(* Logix 5000 project; controller simObli1_rev_1 Emulate 5570 rev 32.11; software revision 32.02 *)

TASK MainTask (continuous, watchdog 500 ms) : MainProgram, Alarmer, MS1_2_Function
TASK simulering (periodic, rate 10 ms, priority 10, watchdog 500 ms) : mainSim
TASK Temp_regulering (periodic, rate 100 ms, priority 10, watchdog 500 ms) : Heat_reg
TASK Tryk_regulering (periodic, rate 500 ms, priority 10, watchdog 500 ms) : Tryk_regulering_PID

MODULES
   Local : Emulate 5570 (ICP 3, rev 32.11)
END_MODULES

TYPE SP :   // De forskellige setpunkter
STRUCT
   Tryk : REAL;   // Tryk regulering
END_STRUCT
END_TYPE

ADD_ON_INSTRUCTION Add_three_Numbers   (* revision 1.0 *)
VAR_INPUT
   nr1 : REAL; {required}
   nr2 : REAL; {required}
   nr3 : REAL; {required}
END_VAR
VAR_OUTPUT
   nr4 : REAL; {access Read Only, required}
END_VAR
VAR
   ADD_01 : FBD_MATH; {access None}
   ADD_02 : FBD_MATH; {access None}
   __l3847ED3F9690BCDD : REAL; {access None}
   __lAC4B0D8890163B21 : REAL; {access None}
   __l5BA8AF029BD9C521 : REAL; {access None}
END_VAR

ROUTINE Logic   (* function block diagram *)
   SHEET 1
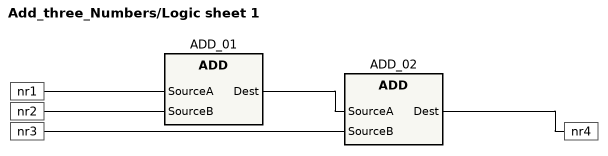
   ADD_01 : ADD(SourceA := nr1, SourceB := nr2);
   ADD_02 : ADD(SourceA := ADD_01.Dest, SourceB := nr3);
   nr4 := ADD_02.Dest;
END_ROUTINE
END_ADD_ON_INSTRUCTION

ADD_ON_INSTRUCTION IMC_Sim   (* revision 1.0 *)
VAR_INPUT
   IMC_CV : REAL; {required}
   IMC_Sim_Reset : BOOL;
   PosNegGain : BOOL;
   DeadTime : REAL := 40.0;
   Lag1 : REAL := 20.0;
   Lag2 : REAL := 20.0;
END_VAR
VAR_OUTPUT
   IMC_PV : REAL; {access Read Only, required}
END_VAR
VAR
   LDLG_01 : LEAD_LAG := (Lag := 30.0, Gain := 1.0, RTSTime := 1);
   LDLG_02 : LEAD_LAG := (Lag := 5.0, Gain := 1.0, RTSTime := 1);
   DEDT_01 : DEADTIME := (Deadtime := 5.0, Gain := 1.0, RTSTime := 1);
   DAIMC : REAL[500];
   SEL_01 : SELECT := (In1 := 1.0, In2 := -1.0);
   SUB_01 : FBD_MATH := (SourceA := 100.0);
   __l19C25824DC418C7C : REAL; {access None}
   __l063CFE09B5704E10 : REAL; {access None}
   __l53C0B5411D4AFA12 : BOOL; {access None}
   __l688BFD8304F18446 : REAL; {access None}
   __l9A341ECD8A034AB4 : REAL; {access None}
   __l887D6C7A4353A221 : BOOL; {access None}
END_VAR

ROUTINE Logic   (* function block diagram *)
   SHEET 1
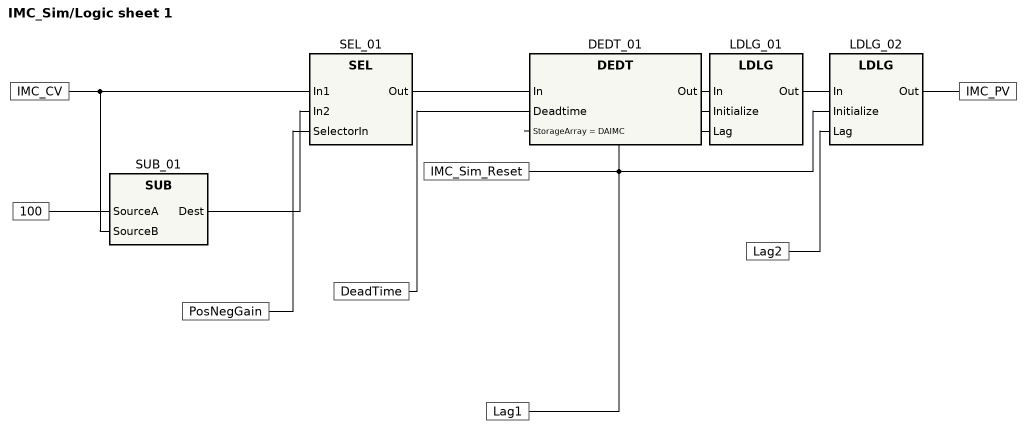
   SUB_01 : SUB(SourceA := 100, SourceB := IMC_CV);
   SEL_01 : SEL(In1 := IMC_CV, In2 := SUB_01.Dest, SelectorIn := PosNegGain);
   DEDT_01 : DEDT(In := SEL_01.Out, Deadtime := DeadTime, StorageArray := DAIMC);
   LDLG_01 : LDLG(In := DEDT_01.Out, Initialize := IMC_Sim_Reset, Lag := Lag1);
   LDLG_02 : LDLG(In := LDLG_01.Out, Initialize := IMC_Sim_Reset, Lag := Lag2);
   IMC_PV := LDLG_02.Out;
END_ROUTINE
END_ADD_ON_INSTRUCTION

ADD_ON_INSTRUCTION Invers_Direkte   (* revision 1.0 *)
VAR_INPUT
   PV : REAL; {required}
   SP : REAL; {required}
END_VAR
VAR_OUTPUT
   fejl_e : REAL; {access None, visible}
END_VAR
VAR_INPUT
   Invers_Direkte : BOOL; {access None, required}
END_VAR
VAR
   SUB_01 : FBD_MATH; {access None}
   SUB_02 : FBD_MATH; {access None}
   SEL_01 : SELECT; {access None}
   Invers : FBD_MATH; {access None}
   Direkte : FBD_MATH; {access None}
   __lF2B22BFB3DCEA4AD : BOOL; {access None}
   __l05D6903D8B432843 : REAL; {access None}
   __lC89B16A93BBA0745 : REAL; {access None}
END_VAR

ROUTINE Logic   (* function block diagram *)
   SHEET 1
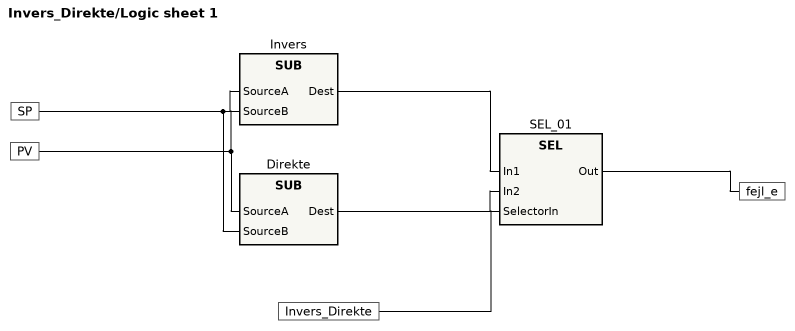
   Invers : SUB(SourceA := SP, SourceB := PV);
   Direkte : SUB(SourceA := PV, SourceB := SP);
   SEL_01 : SEL(In1 := Invers.Dest, In2 := Direkte.Dest, SelectorIn := Invers_Direkte);
   fejl_e := SEL_01.Out;
END_ROUTINE
END_ADD_ON_INSTRUCTION

ADD_ON_INSTRUCTION PID_regulator   (* revision 1.0 *)
VAR_INPUT
   SP : REAL; {access None, visible}
   PV : REAL; {access None, visible}
   Kp : REAL; {access None, visible}
   Ki : REAL; {access None, visible}
   Kd : REAL; {visible}
   U0 : REAL; {visible}
   U_man : REAL; {visible}
END_VAR
VAR_OUTPUT
   CV : REAL; {access Read Only, visible}
END_VAR
VAR_INPUT
   Invers_Direkte : BOOL; {access None, visible}
   Manuel_Auto : BOOL; {access None, visible}
   Reset : BOOL; {visible}
END_VAR
VAR
   Add_three_Numbers_01 : Add_three_Numbers; {access None}
   Invers_Direkte_01 : Invers_Direkte; {access None}
   ADD_02 : FBD_MATH := (SourceA := 23.71752, Dest := 23.71752);
   DERV_01 : DERIVATIVE := (Gain := 5.0, RTSTime := 1, DeltaT := 0.1);
   INTG_01 : INTEGRATOR := (IGain := 4.0, HighLimit := 100.0, LowLimit := -100.0, RTSTime := 1, Out := 23.717138, DeltaT := 0.1);
   MUL_01 : FBD_MATH := (SourceB := 21.5);
   SEL_01 : SELECT;
   Zero : REAL; {access None}
   EQU_01 : FBD_COMPARE; {access None}
   BOR_01 : FBD_BOOLEAN_OR; {access None}
   __l96318BC379C30533 : BOOL; {access None}
   __l2F473B8535F47B00 : REAL; {access None}
   __lA761870FE80B05BE : REAL; {access None}
   __l9EC96B4B26C0C36B : REAL; {access None}
   __lFDE2B6EA02C4DFCD : BOOL; {access None}
   __l4290A7EC9081AB39 : REAL; {access None}
   __l00D9322ED4A60604 : REAL; {access None}
   __l72C6A0FC54AFEFC8 : REAL; {access None}
   __l1ED7CA2F7341DD57 : REAL; {access None}
   __l95CCFAC39C43494D : REAL; {access None}
   __l28D609EBC2B6453D : BOOL; {access None}
END_VAR

ROUTINE Logic   (* function block diagram *)
   SHEET 1
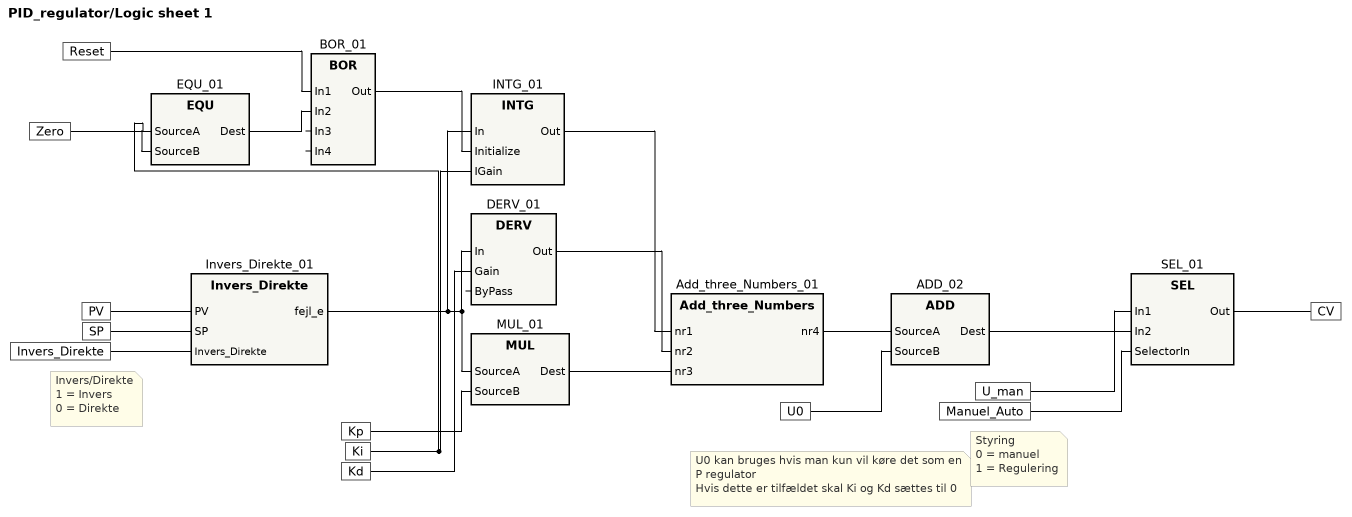
   // Invers/Direkte
   // 1 = Invers
   // 0 = Direkte
   Invers_Direkte_01 : Invers_Direkte(PV := PV, SP := SP, Invers_Direkte := Invers_Direkte);
   EQU_01 : EQU(SourceA := Ki, SourceB := Zero);
   BOR_01 : BOR(In1 := Reset, In2 := EQU_01.Dest);   // unwired pins: In3 In4
   INTG_01 : INTG(In := Invers_Direkte_01.fejl_e, Initialize := BOR_01.Out, IGain := Ki);
   DERV_01 : DERV(In := Invers_Direkte_01.fejl_e, Gain := Kd);   // unwired pins: ByPass
   MUL_01 : MUL(SourceA := Invers_Direkte_01.fejl_e, SourceB := Kp);
   Add_three_Numbers_01 : Add_three_Numbers(nr1 := INTG_01.Out, nr2 := DERV_01.Out, nr3 := MUL_01.Dest);
   // U0 kan bruges hvis man kun vil køre det som en
   // P regulator
   // Hvis dette er tilfældet skal Ki og Kd sættes til 0
   ADD_02 : ADD(SourceA := Add_three_Numbers_01.nr4, SourceB := U0);
   // Styring
   // 0 = manuel
   // 1 = Regulering
   SEL_01 : SEL(In1 := U_man, In2 := ADD_02.Dest, SelectorIn := Manuel_Auto);
   CV := SEL_01.Out;
END_ROUTINE
END_ADD_ON_INSTRUCTION

ADD_ON_INSTRUCTION SplitRange_sim   (* revision 1.1 *)
// Split-Range simulator
VAR_INPUT
   CV_HEAT : REAL; {required}   // Heating signal - aktiv hvis temperature er under SP
   CV_COOL : REAL; {required}   // aktiv hvis temperature er over SP
   Udetemp : REAL; {required}   // Udetemperature - belastning
END_VAR
VAR_OUTPUT
   PV : REAL; {access None, required}   // PV - den målte temperature
   Aktuel_belastning : REAL; {access Read Only}   // Viser den aktuelle belastning
END_VAR
VAR
   ADD_01 : FBD_MATH;
   IMC_Sim_01 : IMC_Sim := (DeadTime := 2.0, Lag1 := 4.0, Lag2 := 4.0, IMC_PV := 0.0004592548);
   LDLG_01 : LEAD_LAG := (In := 1.0, Lag := 4.0, Gain := 1.0, RTSTime := 1, Out := 0.9998808, DeltaT := 0.001);
   SCL_01 : SCALE := (InRawMax := 100.0, InEUMax := -50.0);
   SCL_02 : SCALE := (InRawMax := 100.0, InEUMax := 50.0);
   SUB_100 : FBD_MATH := (SourceA := 100.0, Dest := 100.0);
   SCL_1 : SCALE := (InRawMax := 100.0, InEUMax := -50.0, Limiting := 1); {access None}
   SCL_2 : SCALE := (InRawMax := 100.0, InEUMax := 75.0, Limiting := 1); {access None}
   SUB_01 : FBD_MATH; {access None}
   SCL_03 : SCALE := (InRawMax := 40.0, InRawMin := -20.0, InEUMax := 40.0, InEUMin := -20.0, Limiting := 1); {access None}
   LDLG_02 : LEAD_LAG := (In := 1.0, Lag := 4.0, Gain := 1.0, RTSTime := 1, Out := 0.9998808, DeltaT := 0.001);
   ADD_02 : FBD_MATH; {access None}
   SEL_01 : SELECT := (In1 := 22.0, In2 := 25.0, Out := 22.0); {access None}
   BOR_01 : FBD_BOOLEAN_OR; {access None}
   GEQ_01 : FBD_COMPARE := (SourceA := 22.0, SourceB := 76.0); {access None}
   LEQ_01 : FBD_COMPARE := (SourceA := 22.0, SourceB := -26.0); {access None}
   MSK_Udetemp_lokal : REAL; {access None}   // Lokal Tag
   __l3E8D71CFCB07E059 : REAL; {access None}
   __lE2050592453F5B65 : REAL; {access None}
   __l9DC1ED918EA552ED : REAL; {access None}
   __l5879EB8504FFCE46 : REAL; {access None}
END_VAR

ROUTINE Logic   (* function block diagram *)
   SHEET 1
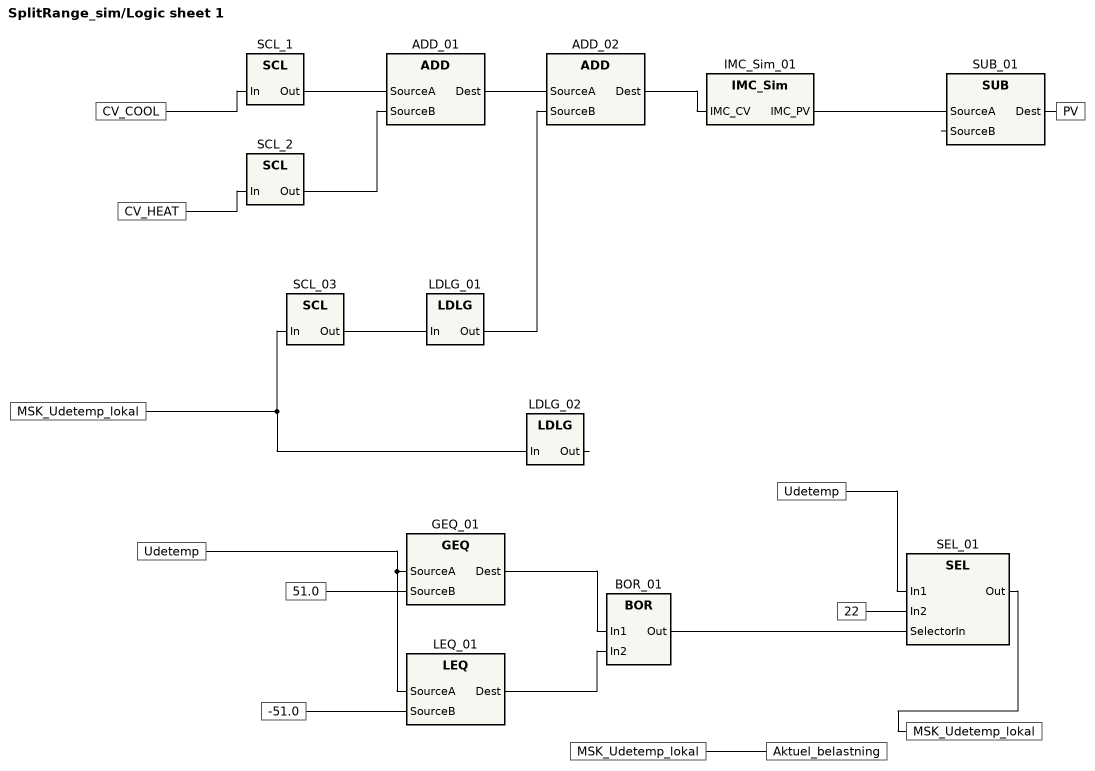
   SCL_1 : SCL(In := CV_COOL);
   SCL_2 : SCL(In := CV_HEAT);
   SCL_03 : SCL(In := MSK_Udetemp_lokal);
   ADD_01 : ADD(SourceA := SCL_1.Out, SourceB := SCL_2.Out);
   GEQ_01 : GEQ(SourceA := Udetemp, SourceB := 51.0);
   LEQ_01 : LEQ(SourceA := Udetemp, SourceB := -51.0);
   LDLG_01 : LDLG(In := SCL_03.Out);
   LDLG_02 : LDLG(In := MSK_Udetemp_lokal);   // unwired pins: Out
   ADD_02 : ADD(SourceA := ADD_01.Dest, SourceB := LDLG_01.Out);
   BOR_01 : BOR(In1 := GEQ_01.Dest, In2 := LEQ_01.Dest);
   IMC_Sim_01 : IMC_Sim(IMC_CV := ADD_02.Dest);
   Aktuel_belastning := MSK_Udetemp_lokal;
   SEL_01 : SEL(In1 := Udetemp, In2 := 22, SelectorIn := BOR_01.Out);
   MSK_Udetemp_lokal := SEL_01.Out;
   SUB_01 : SUB(SourceA := IMC_Sim_01.IMC_PV);   // unwired pins: SourceB
   PV := SUB_01.Dest;
END_ROUTINE
END_ADD_ON_INSTRUCTION

ADD_ON_INSTRUCTION Tryk_simulering   (* revision 1.0, vendor JPJohansen  *)
// Til obligatorisk opgave 1 - PA3
// Revision note:
// ændringer på dødtid og tidskonstant samt navn. den
VAR_INPUT
   Regulator_Ind : REAL; {required}   // CV fra regulatoren 0-100
   belastning : REAL; {visible}
   DeadTime : REAL := 2.0;   // Dødtid 0.1 til 1.99 sek.
   Tidskonstant : REAL := 25.0;   // Tidskonstant i LeadLag 0.1 til 40.0 sek
END_VAR
VAR_OUTPUT
   Tryk_PV : REAL; {access Read Only, required}   // Rumtemperatur i restaurant'en
END_VAR
VAR
   DEDT_01 : DEADTIME := (Gain := 1.0, RTSTime := 1);
   ADD_01 : FBD_MATH;
   LDLG_01 : LEAD_LAG := (Gain := 1.0, RTSTime := 1);
   Gem : REAL[200];
   HLL_01 : HL_LIMIT := (HighLimit := 100.0);
   SCL_01 : SCALE := (InRawMax := 100.0, InEUMax := 10.0, Limiting := 1); {access None}
   __lECFF871F8574D89C : REAL; {access None}
   __l5F788AB00BA17BE2 : REAL; {access None}
   __l383B518581B97AFE : REAL; {access None}
   __l720CE79138866EFB : REAL; {access None}
END_VAR

ROUTINE Logic   (* function block diagram *)
   SHEET 1
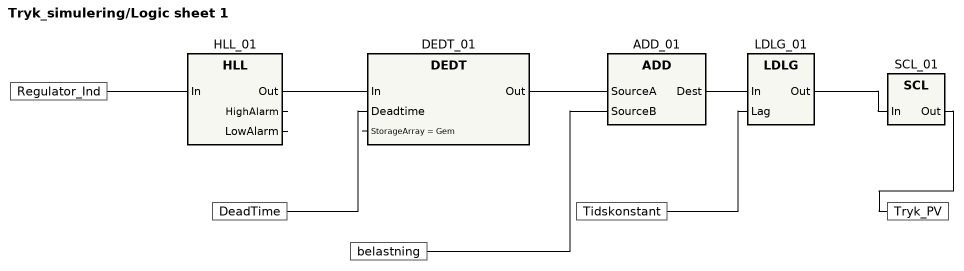
   HLL_01 : HLL(In := Regulator_Ind);   // unwired pins: HighAlarm LowAlarm
   DEDT_01 : DEDT(In := HLL_01.Out, Deadtime := DeadTime, StorageArray := Gem);
   ADD_01 : ADD(SourceA := DEDT_01.Out, SourceB := belastning);
   LDLG_01 : LDLG(In := ADD_01.Dest, Lag := Tidskonstant);
   SCL_01 : SCL(In := LDLG_01.Out);
   Tryk_PV := SCL_01.Out;
END_ROUTINE
END_ADD_ON_INSTRUCTION

VAR_GLOBAL   (* controller tags *)
   Absorbering_MS2 : SFC_STEP := (Status := 16#0820_0001, DN := 1, PauseTimer := 1, T := 34045, TMax := 34045, Count := 12);   // Absorbering_MS2
   AC_1 : BOOL;
   drift : BOOL;
   H1_opvarmer : BOOL;
   Heat_Alarm_Pressure_reduction_step : BOOL;
   Heat_SP : REAL := 5.0;
   Kd : REAL;
   Ki : REAL := 1.0;
   Kp : REAL := 10.0;
   Man_auto : BOOL := 1;
   P_1 : BOOL;
   P_2 : BOOL;
   PT_100 : REAL := 1.523409;
   PT_101 : REAL := 1.77;
   PT_102 : REAL;
   Ready_to_start : BOOL;
   Ready_to_start_step : SFC_STEP := (Status := 16#a820_0201, X := 1, SA := 1, DN := 1, PauseTimer := 1, T := 204423, TMax := 204423, Count := 1);
   Shutdown_valves_step : SFC_STEP := (Status := 16#0020_0001, PauseTimer := 1);
   Sp : REAL := 3.0;
   Standby : SFC_STEP := (Status := 16#0020_0000, PauseTimer := 1);
   start : BOOL;
   stop : BOOL;
   Temp_FF0 : REAL := 22.0;
   Temp_Kd : REAL := 0.03;
   Temp_Kf : REAL;
   Temp_Ki : REAL := 13.2;
   Temp_Kp : REAL := 2.1;
   Temp_Timer : TIMER := (PRE := 10000);
   Temp_Toggle_Timer : BOOL := 1;
   Tran_008 : BOOL;
   TT_100 : REAL := 22.0;
   TT_101 : REAL := 9.999999;
   TT_102 : REAL := -11.000001;
   TT_103 : REAL := 20.064066;
   U_before_split : REAL;
   V_100 : REAL;
   V_101 : BOOL;
   V_102 : BOOL;
   V_103 : BOOL;
   V_104 : BOOL;
   V_105 : REAL;
   V_106 : REAL;
   V_107 : BOOL;
   V_108 : BOOL;
   V_11 : BOOL;
   V_12 : BOOL;
   V_13 : BOOL;
   V_14 : BOOL;
   Valves_off : BOOL;
   VMan_101 : BOOL;
   VMan_102 : BOOL;
   VMan_103 : BOOL;
   VMan_104 : BOOL;
   VMan_107 : BOOL;
   VMan_108 : BOOL;
   VMan_11 : BOOL;
   VMan_12 : BOOL;
   VMan_13 : BOOL;
   VMan_14 : BOOL;
END_VAR

PROGRAM Alarmer   (* main routine Alarm_systemer *)
VAR
   ABS_01 : FBD_MATH_ADVANCED := (Source := 15.067879, Dest := 15.067879);
   GRT_3deg : FBD_COMPARE := (SourceA := 15.067879, SourceB := 3.0, Dest := 1);
   SUB_01 : FBD_MATH := (SourceA := 20.067879, SourceB := 5.0, Dest := 15.067879);
END_VAR

ROUTINE Alarm_systemer   (* ladder *)
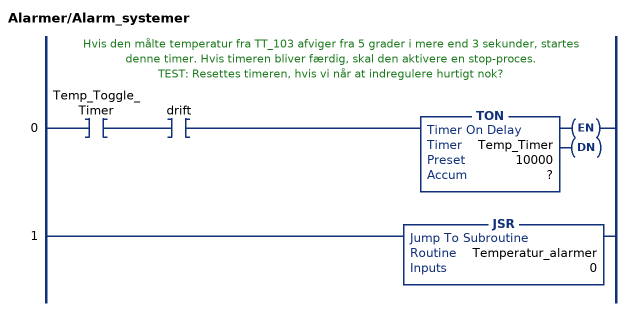
   // Hvis den målte temperatur fra TT_103 afviger fra 5 grader i mere end 3 sekunder, startes denne timer. Hvis timeren bliver færdig, skal den aktivere en stop-proces.
   // TEST: Resettes timeren, hvis vi når at indregulere hurtigt nok?
   0: XIC(Temp_Toggle_Timer)XIC(drift)TON(Temp_Timer,?,?);
   1: JSR(Temperatur_alarmer,0);
END_ROUTINE

ROUTINE Temperatur_alarmer   (* function block diagram *)
   SHEET 1
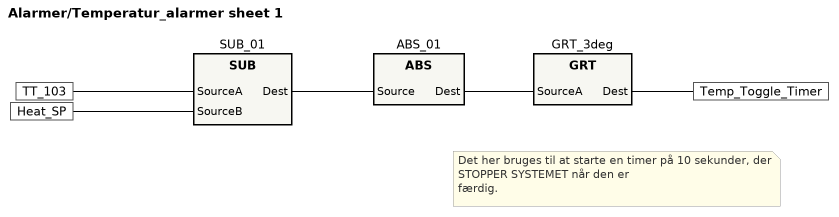
   // Det her bruges til at starte en timer på 10 sekunder, der STOPPER SYSTEMET når den er
   // færdig.
   SUB_01 : SUB(SourceA := TT_103, SourceB := Heat_SP);
   ABS_01 : ABS(Source := SUB_01.Dest);
   GRT_3deg : GRT(SourceA := ABS_01.Dest);
   Temp_Toggle_Timer := GRT_3deg.Dest;
END_ROUTINE
END_PROGRAM

PROGRAM Heat_reg   (* main routine Heat_PIDE *)
VAR
   ADD_01 : FBD_MATH;
   AT_heat : PIDE_AUTOTUNE;
   Auto : BOOL := 1;
   BNOT_01 : FBD_BOOLEAN_NOT := (In := 1);
   GRT_01 : FBD_COMPARE;
   MUL_01 : FBD_MATH;
   needscooling : FBD_COMPARE;
   needsheating : FBD_COMPARE;
   SEL_01 : SELECT := (In1 := 50.0, Out := 50.0);
   SplitCV : SPLIT_RANGE := (In := 50.0, CycleTime := 1.0, MaxHeatIn := 100.0, MinHeatIn := 50.0, MinCoolIn := 50.0, MaxHeatTime := 1.0, MaxCoolTime := 1.0);
   SUB_01 : FBD_MATH := (SourceA := 22.0, SourceB := 22.0);
   TC_PIDE : PID_ENHANCED := (PV := 20.044895, PVEUMax := 100.0, SPOper := 5.0, SPHLimit := 100.0, RatioProg := 1.0, RatioOper := 1.0, RatioHLimit := 1.0, RatioLLimit := 1.0, CVEUMax := 100.0, CVHLimit := 100.0, PGain := 2.1, IGain := 13.2, DGain := 0.03, PVEDerivative := 1, RTSTime := 1, CVLAlarm := 1, SP := 5.0, SPPercent := 5.0, PVPercent := 20.044895, E := -15.044895, EPercent := -15.044895, InitPrimary := 1, WindupLOut := 1, Ratio := 1.0, Auto := 1, DeltaT := 0.1);
   Temp_Timer : BOOL;
   U_heat_manuel : REAL;
END_VAR

ROUTINE Heat_PIDE   (* function block diagram *)
   SHEET 1
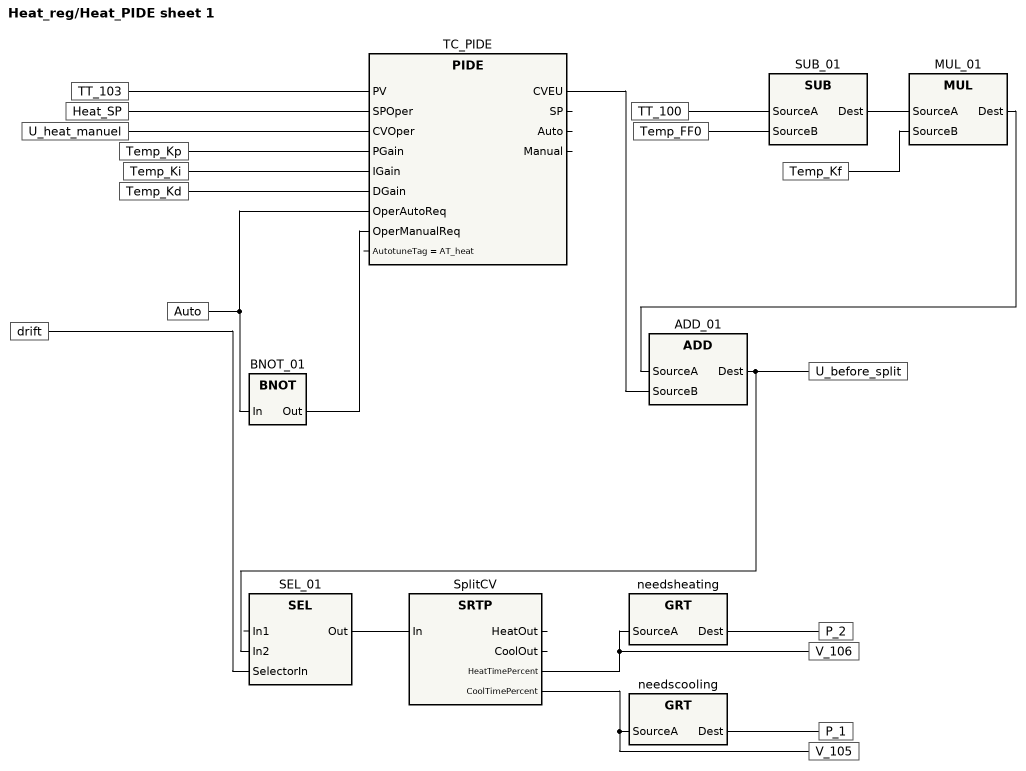
   BNOT_01 : BNOT(In := Auto);
   TC_PIDE : PIDE(PV := TT_103, SPOper := Heat_SP, CVOper := U_heat_manuel, PGain := Temp_Kp, IGain := Temp_Ki, DGain := Temp_Kd, OperAutoReq := Auto, OperManualReq := BNOT_01.Out, AutotuneTag := AT_heat);   // unwired pins: SP Auto Manual
   SUB_01 : SUB(SourceA := TT_100, SourceB := Temp_FF0);
   MUL_01 : MUL(SourceA := SUB_01.Dest, SourceB := Temp_Kf);
   ADD_01 : ADD(SourceA := MUL_01.Dest, SourceB := TC_PIDE.CVEU);
   SEL_01 : SEL(In2 := ADD_01.Dest, SelectorIn := drift);   // unwired pins: In1
   SplitCV : SRTP(In := SEL_01.Out);   // unwired pins: HeatOut CoolOut
   needsheating : GRT(SourceA := SplitCV.HeatTimePercent);
   needscooling : GRT(SourceA := SplitCV.CoolTimePercent);
   U_before_split := ADD_01.Dest;
   V_106 := SplitCV.HeatTimePercent;
   V_105 := SplitCV.CoolTimePercent;
   P_2 := needsheating.Dest;
   P_1 := needscooling.Dest;
END_ROUTINE
END_PROGRAM

PROGRAM MainProgram   (* main routine mainLadder *)

ROUTINE Aux_systems   (* ladder *)
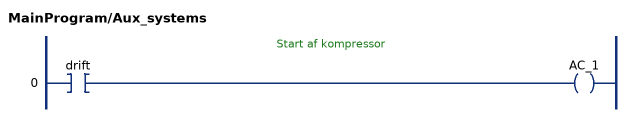
   // Start af kompressor
   0: XIC(drift)OTE(AC_1);
END_ROUTINE

ROUTINE mainLadder   (* ladder *)
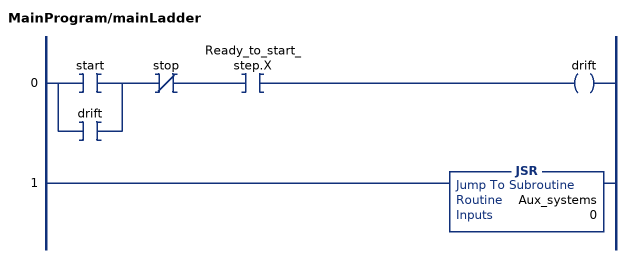
   0: [XIC(start) ,XIC(drift) ]XIO(stop)XIC(Ready_to_start_step.X)OTE(drift);
   1: JSR(Aux_systems,0);
END_ROUTINE
END_PROGRAM

PROGRAM mainSim   (* main routine mainRutine *)
VAR
   BAND_01 : FBD_BOOLEAN_AND := (In3 := 1, In4 := 1, In5 := 1, In6 := 1, In7 := 1, In8 := 1);
   BAND_02 : FBD_BOOLEAN_AND := (In4 := 1, In5 := 1, In6 := 1, In7 := 1, In8 := 1);
   BAND_03 : FBD_BOOLEAN_AND := (In2 := 1, In4 := 1, In5 := 1, In6 := 1, In7 := 1, In8 := 1);
   BAND_04 : FBD_BOOLEAN_AND := (In2 := 1, In4 := 1, In5 := 1, In6 := 1, In7 := 1, In8 := 1);
   BAND_05 : FBD_BOOLEAN_AND := (In4 := 1, In5 := 1, In6 := 1, In7 := 1, In8 := 1);
   BAND_06 : FBD_BOOLEAN_AND := (In3 := 1, In4 := 1, In5 := 1, In6 := 1, In7 := 1, In8 := 1);
   BAND_07 : FBD_BOOLEAN_AND := (In2 := 1, In3 := 1, In4 := 1, In5 := 1, In6 := 1, In7 := 1, In8 := 1);
   BAND_08 : FBD_BOOLEAN_AND := (In3 := 1, In4 := 1, In5 := 1, In6 := 1, In7 := 1, In8 := 1);
   BNOT_01 : FBD_BOOLEAN_NOT := (Out := 1);
   BNOT_02 : FBD_BOOLEAN_NOT := (Out := 1);
   CTUD_01 : FBD_COUNTER := (PRE := 220, ACC := 59);
   CTUD_02 : FBD_COUNTER := (PRE := 220);
   CTUD_03 : FBD_COUNTER := (PRE := 10, ACC := 40, DN := 1);
   CTUD_04 : FBD_COUNTER := (PRE := 10, ACC := 26, DN := 1);
   MS1_koling_OK : BOOL;
   MS1_opvarming_OK : BOOL;
   MS1_trykreduktion_OK : BOOL;
   MS1_trykstigning_OK : BOOL;
   MS2_koling_OK : BOOL;
   MS2_opvarming_OK : BOOL;
   MS2_trykreduktion_OK : BOOL;
   MS2_trykstigning_OK : BOOL;
   SCL_01 : SCALE := (In := 59.0, InRawMax := 100.0, InEUMax := 3.0, Limiting := 1, Out := 1.77);
   SCL_02 : SCALE := (InRawMax := 100.0, InEUMax := 3.0, Limiting := 1);
   SCL_03 : SCALE := (In := 40.0, InRawMax := 100.0, InEUMax := 100.0, InEUMin := -50.0, Limiting := 1, Out := 9.999999);
   SCL_04 : SCALE := (In := 26.0, InRawMax := 100.0, InEUMax := 100.0, InEUMin := -50.0, Limiting := 1, Out := -11.000001);
   SEL_01 : SELECT;
   SEL_02 : SELECT;
   SplitRange_sim_01 : SplitRange_sim := (Udetemp := 22.0, PV := 20.08684, Aktuel_belastning := 22.0);
   TONR_01 : FBD_TIMER := (PRE := 250);
   TONR_02 : FBD_TIMER := (PRE := 250);
   TONR_03 : FBD_TIMER := (PRE := 250);
   TONR_04 : FBD_TIMER := (PRE := 250);
   TONR_05 : FBD_TIMER := (PRE := 350);
   TONR_06 : FBD_TIMER := (PRE := 500);
   TONR_07 : FBD_TIMER := (PRE := 350);
   TONR_08 : FBD_TIMER := (PRE := 500);
   Tryk_simulering_01 : Tryk_simulering := (DeadTime := 2.0, Tidskonstant := 25.0, Tryk_PV := 1.520366);
END_VAR

ROUTINE mainRutine   (* ladder *)
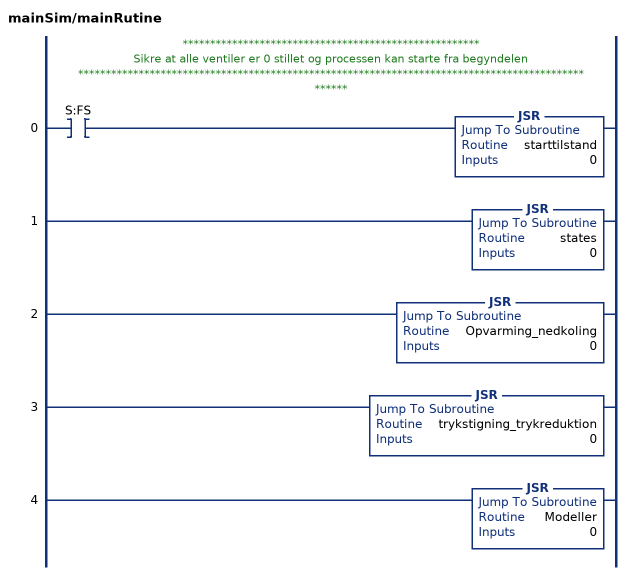
   // ******************************************************
   // Sikre at alle ventiler er 0 stillet og processen kan starte fra begyndelen
   // **************************************************************************************************
   0: XIC(S:FS)JSR(starttilstand,0);
   1: JSR(states,0);
   2: JSR(Opvarming_nedkoling,0);
   3: JSR(trykstigning_trykreduktion,0);
   4: JSR(Modeller,0);
END_ROUTINE

ROUTINE Modeller   (* function block diagram *)
   SHEET 1
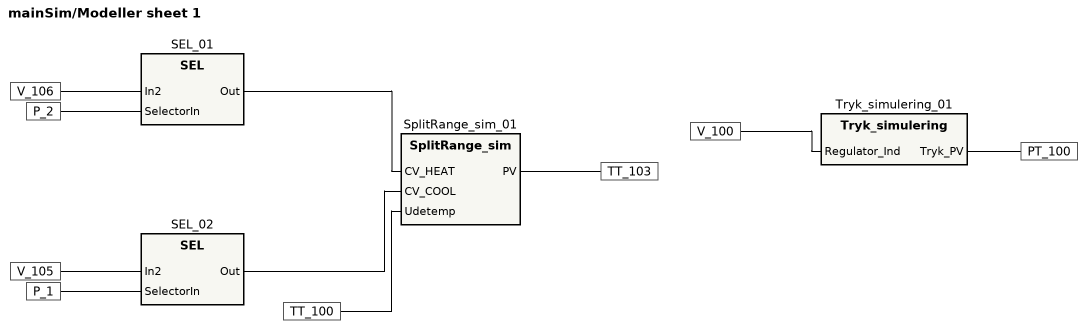
   SEL_01 : SEL(In2 := V_106, SelectorIn := P_2);
   SEL_02 : SEL(In2 := V_105, SelectorIn := P_1);
   SplitRange_sim_01 : SplitRange_sim(CV_HEAT := SEL_01.Out, CV_COOL := SEL_02.Out, Udetemp := TT_100);
   TT_103 := SplitRange_sim_01.PV;
   Tryk_simulering_01 : Tryk_simulering(Regulator_Ind := V_100);
   PT_100 := Tryk_simulering_01.Tryk_PV;
END_ROUTINE

ROUTINE Opvarming_nedkoling   (* function block diagram *)
   SHEET 1
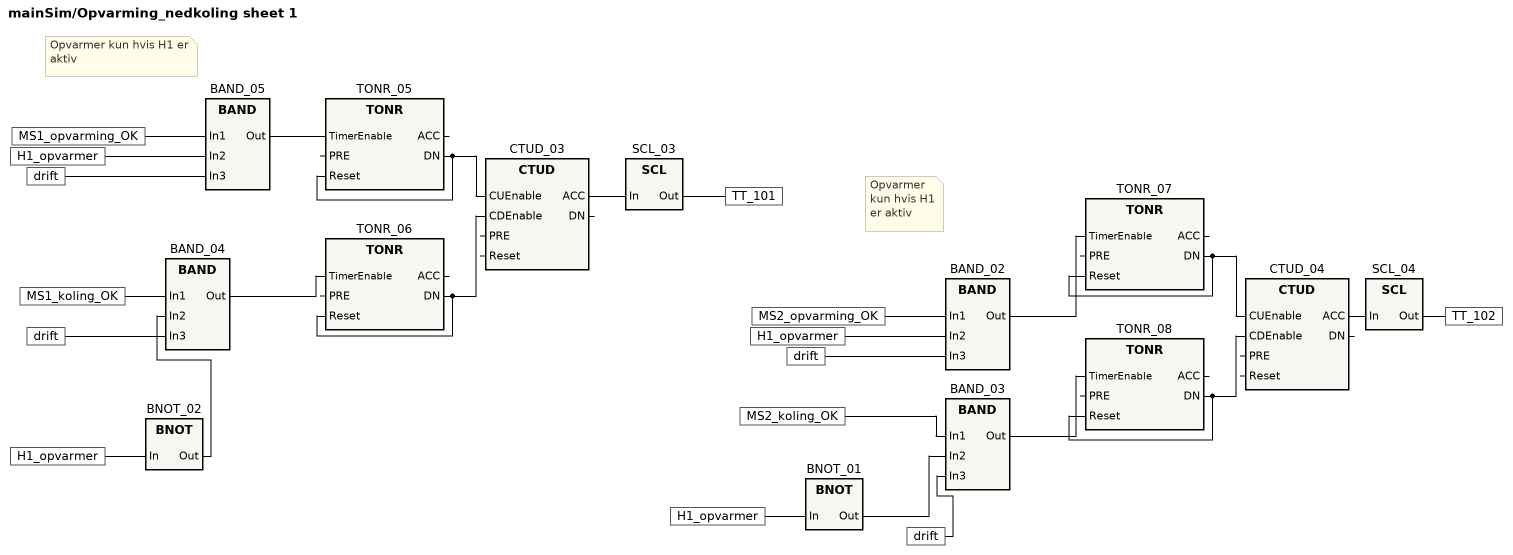
   // Opvarmer kun hvis H1 er
   // aktiv
   BNOT_02 : BNOT(In := H1_opvarmer);
   BAND_04 : BAND(In1 := MS1_koling_OK, In2 := BNOT_02.Out, In3 := drift);
   BAND_05 : BAND(In1 := MS1_opvarming_OK, In2 := H1_opvarmer, In3 := drift);
   BNOT_01 : BNOT(In := H1_opvarmer);
   // Opvarmer
   // kun hvis H1
   // er aktiv
   BAND_02 : BAND(In1 := MS2_opvarming_OK, In2 := H1_opvarmer, In3 := drift);
   BAND_03 : BAND(In1 := MS2_koling_OK, In2 := BNOT_01.Out, In3 := drift);
   TONR_05 : TONR(TimerEnable := BAND_05.Out, Reset := TONR_05.DN);   // unwired pins: PRE ACC
   TONR_06 : TONR(TimerEnable := BAND_04.Out, Reset := TONR_06.DN);   // unwired pins: PRE ACC
   CTUD_03 : CTUD(CUEnable := TONR_05.DN, CDEnable := TONR_06.DN);   // unwired pins: PRE Reset DN
   SCL_03 : SCL(In := CTUD_03.ACC);
   TT_101 := SCL_03.Out;
   TONR_07 : TONR(TimerEnable := BAND_02.Out, Reset := TONR_07.DN);   // unwired pins: PRE ACC
   TONR_08 : TONR(TimerEnable := BAND_03.Out, Reset := TONR_08.DN);   // unwired pins: PRE ACC
   CTUD_04 : CTUD(CUEnable := TONR_07.DN, CDEnable := TONR_08.DN);   // unwired pins: PRE Reset DN
   SCL_04 : SCL(In := CTUD_04.ACC);
   TT_102 := SCL_04.Out;
END_ROUTINE

ROUTINE starttilstand   (* structured text *)
// Definerer ventilpositioner ved start , First Pass.
   // All valves are closed in First Pass
   // Rutine kan also be run with RESET
   // Globale Tags
   V_11 := 0;
   V_12 := 0;
   V_13 := 0;
   V_14 := 0;
   V_101 := 0;
   V_102 := 0;
   V_103 := 0;
   V_104 := 0;
   V_107 := 0;
   V_108 := 0;
   
END_ROUTINE

ROUTINE states   (* structured text *)
   
   // 4 regeneration steps for each MS
   // Fixed Valve positions for each step - ELSE step not activated
   //*****************************************************************
   // START - Steps for Mole Sieve 1
   // *******************************************************************
   
   IF V_11 and not V_12 and not V_13 and not V_14 and not V_101 and V_102 and not V_103 and V_104 and not V_107 and not V_108 then
   	MS1_trykreduktion_OK := 1;
   else
   	MS1_trykreduktion_OK := 0;
   end_if;
   
   IF V_11 and not V_12 and V_13 and not V_14 and not V_101 and V_102 and not V_103 and V_104 and V_107 and not V_108 then
   	MS1_opvarming_OK := 1;
   else
   	MS1_opvarming_OK := 0;
   end_if;
   
   IF V_11 and not V_12 and V_13 and not V_14 and not V_101 and V_102 and not V_103 and V_104 and not V_107 and V_108 then
   	MS1_koling_OK := 1;
   else
   	MS1_koling_OK := 0;
   end_if;
   
   IF not V_11 and not V_12 and V_13 and not V_14 and not V_101 and V_102 and not V_103 and V_104 and not V_107 and V_108 then
   	MS1_trykstigning_OK := 1;
   else
   	MS1_trykstigning_OK := 0;
   end_if;
   
   
   // END - Steps for Mole Sieve 1
   // *******************************************************************
   // START - Steps for Mole Sieve 2
   // *******************************************************************
   
   IF not V_11 and V_12 and not V_13 and not V_14 and V_101 and not V_102 and V_103 and not V_104 and not V_107 and not V_108 then
   	MS2_trykreduktion_OK := 1;
   else
   	MS2_trykreduktion_OK := 0;
   end_if;
   
   IF not V_11 and V_12 and not V_13 and V_14 and V_101 and not V_102 and V_103 and not V_104 and V_107 and not V_108 then
   	MS2_opvarming_OK := 1;
   else
   	MS2_opvarming_OK := 0;
   end_if;
   
   IF not V_11 and V_12 and not V_13 and V_14 and V_101 and not V_102 and V_103 and not V_104 and not V_107 and V_108 then
   	MS2_koling_OK := 1;
   else
   	MS2_koling_OK := 0;
   end_if;
   
   IF not V_11 and not V_12 and not V_13 and V_14 and V_101 and not V_102 and V_103 and not V_104 and not V_107 and V_108 then
   	MS2_trykstigning_OK := 1;
   else
   	MS2_trykstigning_OK := 0;
   end_if;
   
   // END - Steps for Mole Sieve 2
   // *******************************************************************
END_ROUTINE

ROUTINE trykstigning_trykreduktion   (* function block diagram *)
   SHEET 1
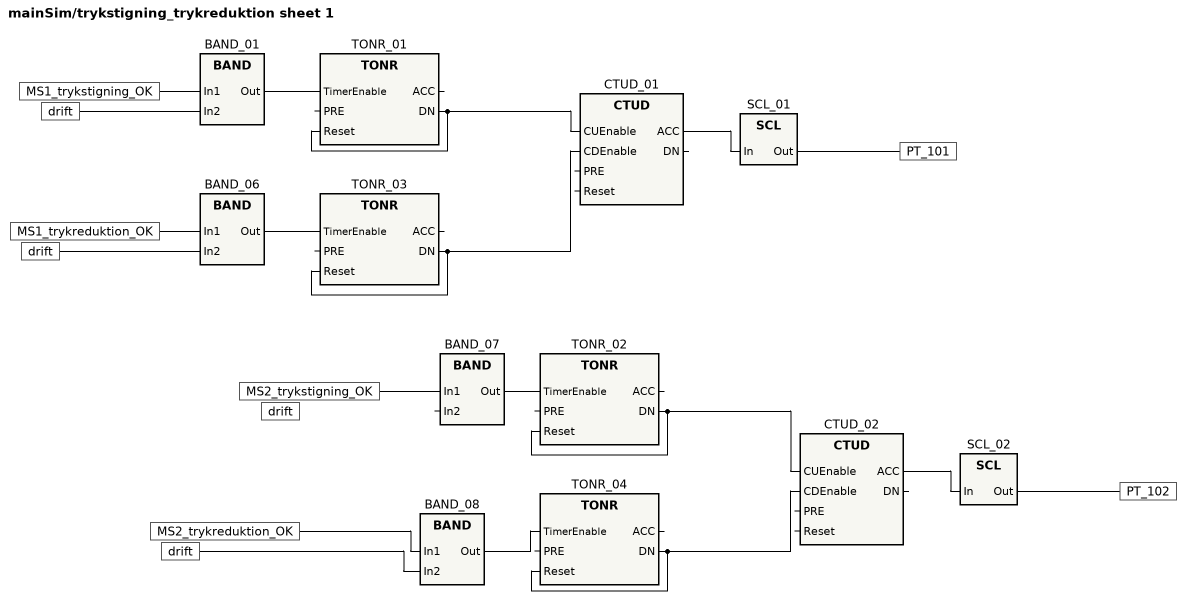
   BAND_01 : BAND(In1 := MS1_trykstigning_OK, In2 := drift);
   BAND_06 : BAND(In1 := MS1_trykreduktion_OK, In2 := drift);
   // unwired input reference drift
   BAND_08 : BAND(In1 := MS2_trykreduktion_OK, In2 := drift);
   BAND_07 : BAND(In1 := MS2_trykstigning_OK);   // unwired pins: In2
   TONR_01 : TONR(TimerEnable := BAND_01.Out, Reset := TONR_01.DN);   // unwired pins: PRE ACC
   TONR_03 : TONR(TimerEnable := BAND_06.Out, Reset := TONR_03.DN);   // unwired pins: PRE ACC
   CTUD_01 : CTUD(CUEnable := TONR_01.DN, CDEnable := TONR_03.DN);   // unwired pins: PRE Reset DN
   SCL_01 : SCL(In := CTUD_01.ACC);
   PT_101 := SCL_01.Out;
   TONR_02 : TONR(TimerEnable := BAND_07.Out, Reset := TONR_02.DN);   // unwired pins: PRE ACC
   TONR_04 : TONR(TimerEnable := BAND_08.Out, Reset := TONR_04.DN);   // unwired pins: PRE ACC
   CTUD_02 : CTUD(CUEnable := TONR_02.DN, CDEnable := TONR_04.DN);   // unwired pins: PRE Reset DN
   SCL_02 : SCL(In := CTUD_02.ACC);
   PT_102 := SCL_02.Out;
END_ROUTINE
END_PROGRAM

PROGRAM MS1_2_Function   (* main routine MS1_Ladder *)
// Main
VAR
   Absorbering_MS1 : SFC_STEP := (Status := 16#0020_0000, PauseTimer := 1);   // Vente step.016 for absorbere Ms.1
   AbsorberingMS1 : SFC_STEP := (Status := 16#0220_0001, AlarmEn := 1, PauseTimer := 1, LimitHigh := 60);   // Absorbering MS-1
   Koeling_MS2 : SFC_STEP := (Status := 16#0020_0001, PauseTimer := 1);   // Køling MS-2 (MS_2 Ladder rung 4 )
   KoelingMS1 : SFC_STEP := (Status := 16#0820_0001, DN := 1, PauseTimer := 1, T := 14132, TMax := 14169, Count := 6);   // Køling MS-1,( MS_1 - Ladder ( rung 8)
   OpvarmningMS1 : SFC_STEP := (Status := 16#0aa0_0001, DN := 1, AlarmEn := 1, AlarmHigh := 1, PauseTimer := 1, T := 8973, TMax := 15278, Count := 12, LimitHigh := 44);   // Opvarmning MS-1, ( MS_1 Ladder - rung 3)
   OpvarmningMS2 : SFC_STEP := (Status := 16#0020_0001, PauseTimer := 1);   // Opvarmning MS-2 (MS_2 Ladder rung 1,2,3 )
   Standby : SFC_STEP := (Status := 16#a820_0201, X := 1, SA := 1, DN := 1, PauseTimer := 1, T := 16821, TMax := 16821, Count := 266);   // Standby
   Step_001 : SFC_STEP := (Status := 16#0020_0000, PauseTimer := 1);   // Trykreduktion MS-2 ( MS_2 Ladder - rung 0 )
   Step_002 : SFC_STEP := (Status := 16#0020_0000, PauseTimer := 1);   // Trykreduktion MS-1 - Ventil V_11 ( MS_1 Ladder - Rung 2)
   Step_009 : SFC_STEP := (Status := 16#0020_0000, PauseTimer := 1);   // Absorbere step
   Step_011 : SFC_STEP := (Status := 16#0020_0000, PauseTimer := 1);
   Step_012 : SFC_STEP := (Status := 16#0020_0000, PauseTimer := 1);
   Step_013 : SFC_STEP := (Status := 16#0020_0000, PauseTimer := 1);
   Step_014 : SFC_STEP := (Status := 16#0020_0000, PauseTimer := 1);
   Step_015 : SFC_STEP := (Status := 16#0020_0000, PauseTimer := 1);
   Tran_000 : BOOL;
   Tran_001 : BOOL;
   Tran_002 : BOOL := 1;
   Tran_003 : BOOL;
   Tran_004 : BOOL := 1;
   Tran_005 : BOOL;
   Tran_006 : BOOL := 1;
   Tran_007 : BOOL;
   Tran_009 : BOOL;
   Tran_010 : BOOL;
   Tran_011 : BOOL;
   Tran_013 : BOOL;
   Tran_014 : BOOL;
   Tran_015 : BOOL;
   TreykreduktionMS2 : SFC_STEP := (Status := 16#0020_0001, PauseTimer := 1);   // Trykreduktion MS-2 ( MS_2 Ladder - rung 0 )
   TrykreduktionMS1 : SFC_STEP := (Status := 16#0820_0001, DN := 1, PauseTimer := 1, T := 23, TMax := 23, Count := 12);   // Trykreduktion MS-1 - Ventil V_11 ( MS_1 Ladder - Rung 2)
   TrykstigningMS1 : SFC_STEP := (Status := 16#0820_0001, DN := 1, PauseTimer := 1, T := 10917, TMax := 10917, Count := 3);   // Trykstigning MS-1, PT_101 skal stige til 2 bar
   TrykstigningMS2 : SFC_STEP := (Status := 16#0020_0001, PauseTimer := 1);   // Trykstigning MS-2
END_VAR

ROUTINE Check_Stop   (* ladder *)
// MainTask --> MS1_2_Function
// Kontrollerer stop-processer, som returnerer os til standby.
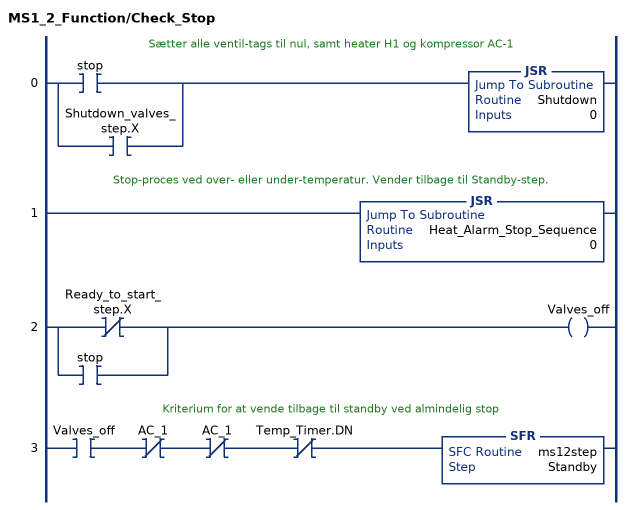
   // Sætter alle ventil-tags til nul, samt heater H1 og kompressor AC-1
   0: [XIC(stop) ,XIC(Shutdown_valves_step.X) ]JSR(Shutdown,0);
   // Stop-proces ved over- eller under-temperatur. Vender tilbage til Standby-step.
   1: JSR(Heat_Alarm_Stop_Sequence,0);
   2: [XIO(Ready_to_start_step.X) ,XIC(stop) ]OTE(Valves_off);
   // Kriterium for at vende tilbage til standby ved almindelig stop
   3: XIC(Valves_off)XIO(AC_1)XIO(AC_1)XIO(Temp_Timer.DN)SFR(ms12step,Standby);
END_ROUTINE

ROUTINE Heat_Alarm_Stop_Sequence   (* sequential function chart *)
// Maintask -> MS1_2_Function
// Shutdown process, pressure relief MS1 and MS2 and then return to standby
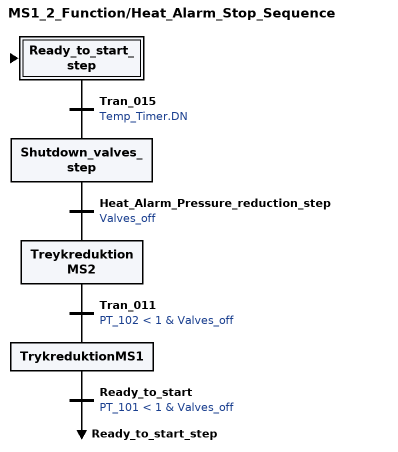
   INITIAL_STEP Ready_to_start_step:
   END_STEP
   TRANSITION Tran_015 FROM Ready_to_start_step TO Shutdown_valves_step
      := Temp_Timer.DN
   END_TRANSITION
   STEP Shutdown_valves_step:
   END_STEP
   TRANSITION Heat_Alarm_Pressure_reduction_step FROM Shutdown_valves_step TO TreykreduktionMS2
      := Valves_off
         
   END_TRANSITION
   STEP TreykreduktionMS2:
   END_STEP
   TRANSITION Tran_011 FROM TreykreduktionMS2 TO TrykreduktionMS1
      := PT_102 < 1 & Valves_off
   END_TRANSITION
   STEP TrykreduktionMS1:
   END_STEP
   TRANSITION Ready_to_start FROM TrykreduktionMS1 TO Ready_to_start_step
      := PT_101 < 1 & Valves_off
   END_TRANSITION
END_ROUTINE

ROUTINE ms12step   (* sequential function chart *)
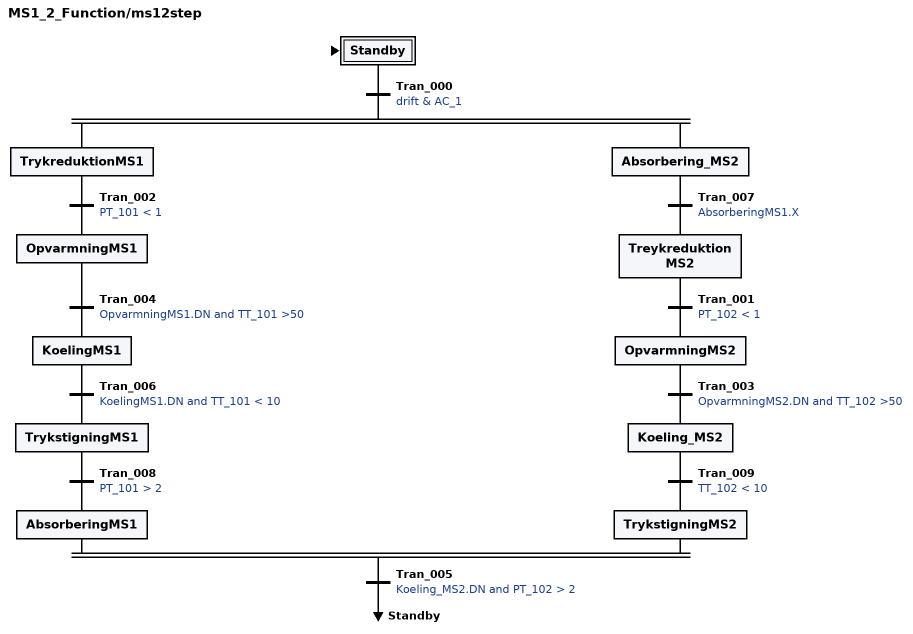
   INITIAL_STEP Standby:
   END_STEP
   TRANSITION Tran_000 FROM Standby TO (TrykreduktionMS1, Absorbering_MS2)
      := drift & AC_1
         
   END_TRANSITION
   STEP TrykreduktionMS1:
   END_STEP
   STEP Absorbering_MS2:
   END_STEP
   TRANSITION Tran_002 FROM TrykreduktionMS1 TO OpvarmningMS1
      := PT_101 < 1
   END_TRANSITION
   TRANSITION Tran_007 FROM Absorbering_MS2 TO TreykreduktionMS2
      := AbsorberingMS1.X
   END_TRANSITION
   STEP OpvarmningMS1:
   END_STEP
   STEP TreykreduktionMS2:
   END_STEP
   TRANSITION Tran_004 FROM OpvarmningMS1 TO KoelingMS1
      := OpvarmningMS1.DN and TT_101 >50
   END_TRANSITION
   TRANSITION Tran_001 FROM TreykreduktionMS2 TO OpvarmningMS2
      := PT_102 < 1
   END_TRANSITION
   STEP KoelingMS1:
   END_STEP
   STEP OpvarmningMS2:
   END_STEP
   TRANSITION Tran_006 FROM KoelingMS1 TO TrykstigningMS1
      := KoelingMS1.DN and
         TT_101 < 10
   END_TRANSITION
   TRANSITION Tran_003 FROM OpvarmningMS2 TO Koeling_MS2
      := OpvarmningMS2.DN and TT_102 >50
         
   END_TRANSITION
   STEP TrykstigningMS1:
   END_STEP
   STEP Koeling_MS2:
   END_STEP
   TRANSITION Tran_008 FROM TrykstigningMS1 TO AbsorberingMS1
      := PT_101 > 2
   END_TRANSITION
   TRANSITION Tran_009 FROM Koeling_MS2 TO TrykstigningMS2
      := TT_102 < 10
   END_TRANSITION
   STEP AbsorberingMS1:
   END_STEP
   STEP TrykstigningMS2:
   END_STEP
   TRANSITION Tran_005 FROM (AbsorberingMS1, TrykstigningMS2) TO Standby
      := Koeling_MS2.DN and PT_102 > 2
   END_TRANSITION
END_ROUTINE
